	(* Internal method *)
	{attribute 'hide'}
	METHOD FB_init : BOOL
	VAR_INPUT
		(*  if TRUE, the retain variables are initialized (warm start / cold start) *)
		bInitRetains : BOOL;
		(*  if TRUE, the instance afterwards gets moved into the copy code (online change) *)
		bInCopyCode : BOOL;
	END_VAR
END_METHOD


	(* Internal method *)
	{attribute 'hide'}
	METHOD FB_exit : BOOL
	VAR_INPUT
		(*  if TRUE, the exit method is called for exiting an instance that is copied afterwards (online change). *)
		bInCopyCode : BOOL;
	END_VAR
END_METHOD


	(* Set the rotation angle in degrees [Â°]. *)
	METHOD SetAngle
	VAR_INPUT
		(* Rotation angle to set in degrees [Â°]. *)
		angle : LREAL;
	END_VAR
END_METHOD


	(* Set the components of this vector to '0.0'. *)
	METHOD SetZero
END_METHOD


	(* Set the components of this orientation. *)
	METHOD SetValues
	VAR_IN_OUT
		(* The position values to set. *)
 {attribute 'GUID' := 'ABCF5F54-5133-060C-4FEE-702387088411'}
				orientation2D : Orientation2D;
	END_VAR
END_METHOD


	(* Get the direction of the local x-axis. *)
	METHOD GetDirectionX
	VAR_IN_OUT
		(* The local x-direction of this orientation. *)
 {attribute 'GUID' := '619D5D7D-53EC-0B73-54D5-FB9C43AFDE82'}
				localX : TangentXY;
	END_VAR
END_METHOD


	(* Get the direction of the local y-axis. *)
	METHOD GetDirectionY
	VAR_IN_OUT
		(* The local y-direction of this orientation. *)
 {attribute 'GUID' := '619D5D7D-53EC-0B73-54D5-FB9C43AFDE82'}
				localY : TangentXY;
	END_VAR
END_METHOD


	(* Invert this position. *)
	METHOD Invert
END_METHOD


	(* Multiply an orientation to this orientation. *)
	METHOD ConcatenateWith
	VAR_IN_OUT
		(* Orientation to concatenate with. *)
 {attribute 'GUID' := 'ABCF5F54-5133-060C-4FEE-702387088411'}
				orientation2D : Orientation2D;
	END_VAR
END_METHOD


	(* Turn the orientation. *)
	METHOD TurnByC
	VAR_INPUT
		(* Rotation angle to turn by in degrees [Â°]. *)
		angle : LREAL;
	END_VAR
END_METHOD


	(* Rotate a PositionXY according to this orientation. *)
	METHOD Transform
	VAR_IN_OUT
		(* The orientation to multipy by. *)
 {attribute 'GUID' := 'D1D75488-37B1-0155-53AF-A9A9BDBB4FFD'}
				positionXY : PositionXY;
	END_VAR
END_METHOD


	PROPERTY angle : LREAL
GET
END_GET
SET
END_SET
END_PROPERTY

END_FUNCTION_BLOCK

// POUs/Spatial/Functions/ConcatenateABC

	{attribute 'TcIecLibraryType'}
	{attribute 'external_name' := 'ConcatenateABC_GUID_5F49A3AF_77BC_0B6E_5B9D_5571A51DBC7B'}
	(* Concatenate two instances of Orientation3D. *)
	FUNCTION ConcatenateABC : BOOL
	VAR_IN_OUT
		rotation0	:	Orientation3D;	(* 1st input orientation of the concatenation. *)
		rotation1	:	Orientation3D;	(* 2nd input orientation of the concatenation. *)
		concatenation	:	Orientation3D;	(* The concatenation of the two input instances. *)
	END_VAR

END_FUNCTION

// POUs/Spatial/Positions/Orientation3D

	{attribute 'c++_compatible'}
	{attribute 'external_name' := 'Orientation3D_GUID_CF039E61_7293_0F6E_5C80_E794F941E4DD'}
	{attribute 'TcIecLibraryType'}
	{attribute 'no_explicit_call' :='do not call this POU directly'}
	{attribute 'no_assign'}
	(* 3D orientation. All angles in degrees [Â°]. *)
	FUNCTION_BLOCK Orientation3D
	VAR
		(* Rotation around the 1st local axis in degrees [Â°]. *)
		p0 : LREAL;
		(* Rotation around 2nd local axis in degrees [Â°]. *)
		p1 : LREAL;
		(* Rotation around 3rd local axis in degrees [Â°]. *)
		p2 : LREAL;
		(* Defines the rotation order (rotate around local axes from left to right) *)
		 {attribute 'GUID' := 'BF8BCC1E-925E-4A57-801C-CC42AFDDA86D'}
		coordinates : E_RotationCoordinates := E_RotationCoordinates.CBA;
		 {attribute 'hide'}
		_reserved1 : ARRAY [1..84] OF USINT;
	END_VAR


	(* Internal method *)
	{attribute 'hide'}
	METHOD FB_init : BOOL
	VAR_INPUT
		(*  if TRUE, the retain variables are initialized (warm start / cold start) *)
		bInitRetains : BOOL;
		(*  if TRUE, the instance afterwards gets moved into the copy code (online change) *)
		bInCopyCode : BOOL;
	END_VAR
END_METHOD


	(* Internal method *)
	{attribute 'hide'}
	METHOD FB_exit : BOOL
	VAR_INPUT
		(*  if TRUE, the exit method is called for exiting an instance that is copied afterwards (online change). *)
		bInCopyCode : BOOL;
	END_VAR
END_METHOD


	(* Set the components of this vector to '0.0'. *)
	METHOD SetZero
END_METHOD


	(* Set the components of this position. *)
	METHOD SetValues
	VAR_IN_OUT
		(* The position values to set. *)
 {attribute 'GUID' := 'CF039E61-7293-0F6E-5C80-E794F941E4DD'}
				orientation3D : Orientation3D;
	END_VAR
END_METHOD


	(* Set the coordinates of the orientation. *)
	METHOD SetValuesABC
	VAR_INPUT
		(* 1st rotation angle in degrees [Â°]. *)
		phi0 : LREAL;
		(* 2nd rotation angle in degrees [Â°]. *)
		phi1 : LREAL;
		(* 3rd rotation angle in degrees [Â°]. *)
		phi2 : LREAL;
	END_VAR
END_METHOD


	(* Set the coordinates of the orientation. *)
	METHOD SetValuesACB
	VAR_INPUT
		(* 1st rotation angle in degrees [Â°]. *)
		phi0 : LREAL;
		(* 2nd rotation angle in degrees [Â°]. *)
		phi1 : LREAL;
		(* 3rd rotation angle in degrees [Â°]. *)
		phi2 : LREAL;
	END_VAR
END_METHOD


	(* Set the coordinates of the orientation. *)
	METHOD SetValuesBCA
	VAR_INPUT
		(* 1st rotation angle in degrees [Â°]. *)
		phi0 : LREAL;
		(* 2nd rotation angle in degrees [Â°]. *)
		phi1 : LREAL;
		(* 3rd rotation angle in degrees [Â°]. *)
		phi2 : LREAL;
	END_VAR
END_METHOD


	(* Set the coordinates of the orientation. *)
	METHOD SetValuesBAC
	VAR_INPUT
		(* 1st rotation angle in degrees [Â°]. *)
		phi0 : LREAL;
		(* 2nd rotation angle in degrees [Â°]. *)
		phi1 : LREAL;
		(* 3rd rotation angle in degrees [Â°]. *)
		phi2 : LREAL;
	END_VAR
END_METHOD


	(* Set the coordinates of the orientation. *)
	METHOD SetValuesCAB
	VAR_INPUT
		(* 1st rotation angle in degrees [Â°]. *)
		phi0 : LREAL;
		(* 2nd rotation angle in degrees [Â°]. *)
		phi1 : LREAL;
		(* 3rd rotation angle in degrees [Â°]. *)
		phi2 : LREAL;
	END_VAR
END_METHOD


	(* Set the coordinates of the orientation. *)
	METHOD SetValuesCBA
	VAR_INPUT
		(* 1st rotation angle in degrees [Â°]. *)
		phi0 : LREAL;
		(* 2nd rotation angle in degrees [Â°]. *)
		phi1 : LREAL;
		(* 3rd rotation angle in degrees [Â°]. *)
		phi2 : LREAL;
	END_VAR
END_METHOD


	(* Set the coordinates of the orientation. *)
	METHOD SetValuesABA
	VAR_INPUT
		(* 1st rotation angle in degrees [Â°]. *)
		phi0 : LREAL;
		(* 2nd rotation angle in degrees [Â°]. *)
		phi1 : LREAL;
		(* 3rd rotation angle in degrees [Â°]. *)
		phi2 : LREAL;
	END_VAR
END_METHOD


	(* Set the coordinates of the orientation. *)
	METHOD SetValuesACA
	VAR_INPUT
		(* 1st rotation angle in degrees [Â°]. *)
		phi0 : LREAL;
		(* 2nd rotation angle in degrees [Â°]. *)
		phi1 : LREAL;
		(* 3rd rotation angle in degrees [Â°]. *)
		phi2 : LREAL;
	END_VAR
END_METHOD


	(* Set the coordinates of the orientation. *)
	METHOD SetValuesBCB
	VAR_INPUT
		(* 1st rotation angle in degrees [Â°]. *)
		phi0 : LREAL;
		(* 2nd rotation angle in degrees [Â°]. *)
		phi1 : LREAL;
		(* 3rd rotation angle in degrees [Â°]. *)
		phi2 : LREAL;
	END_VAR
END_METHOD


	(* Set the coordinates of the orientation. *)
	METHOD SetValuesBAB
	VAR_INPUT
		(* 1st rotation angle in degrees [Â°]. *)
		phi0 : LREAL;
		(* 2nd rotation angle in degrees [Â°]. *)
		phi1 : LREAL;
		(* 3rd rotation angle in degrees [Â°]. *)
		phi2 : LREAL;
	END_VAR
END_METHOD


	(* Set the coordinates of the orientation. *)
	METHOD SetValuesCAC
	VAR_INPUT
		(* 1st rotation angle in degrees [Â°]. *)
		phi0 : LREAL;
		(* 2nd rotation angle in degrees [Â°]. *)
		phi1 : LREAL;
		(* 3rd rotation angle in degrees [Â°]. *)
		phi2 : LREAL;
	END_VAR
END_METHOD


	(* Set the coordinates of the orientation. *)
	METHOD SetValuesCBC
	VAR_INPUT
		(* 1st rotation angle in degrees [Â°]. *)
		phi0 : LREAL;
		(* 2nd rotation angle in degrees [Â°]. *)
		phi1 : LREAL;
		(* 3rd rotation angle in degrees [Â°]. *)
		phi2 : LREAL;
	END_VAR
END_METHOD


	(* Get the direction of the local x-axis. *)
	METHOD GetDirectionX
	VAR_IN_OUT
		(* The local x-direction of this orientation. *)
 {attribute 'GUID' := 'B2E383A0-A70D-05BB-6EF1-4EF1FE579E25'}
				localX : Tangent3D;
	END_VAR
END_METHOD


	(* Get the direction of the local y-axis. *)
	METHOD GetDirectionY
	VAR_IN_OUT
		(* The local y-direction of this orientation. *)
 {attribute 'GUID' := 'B2E383A0-A70D-05BB-6EF1-4EF1FE579E25'}
				localY : Tangent3D;
	END_VAR
END_METHOD


	(* Get the direction of the local z-axis. *)
	METHOD GetDirectionZ
	VAR_IN_OUT
		(* The local z-direction of this orientation. *)
 {attribute 'GUID' := 'B2E383A0-A70D-05BB-6EF1-4EF1FE579E25'}
				localZ : Tangent3D;
	END_VAR
END_METHOD


	(* Invert this position. *)
	METHOD Invert
END_METHOD


	(* Multiply an orientation to this orientation. *)
	METHOD ConcatenateWith
	VAR_IN_OUT
		(* Orientation to concatenate with. *)
 {attribute 'GUID' := 'CF039E61-7293-0F6E-5C80-E794F941E4DD'}
				orientation : Orientation3D;
	END_VAR
END_METHOD


	(* Rotate around an arbitrary local axis. The turn angle is given by the length of the axis. *)
	METHOD TurnBy
	VAR_IN_OUT
		(* The axis of rotation. Its length represents the angle of rotation in degrees [Â°]. *)
 {attribute 'GUID' := '40BB739E-8B51-070D-548D-A1BF22EE7364'}
				axis : TangentABC;
	END_VAR
END_METHOD


	(* Rotation around the local x-axis. *)
	METHOD TurnByA
	VAR_INPUT
		(* The angle to rotate by in degrees [Â°]. *)
		da : LREAL;
	END_VAR
END_METHOD


	(* Rotation around the local y-axis. *)
	METHOD TurnByB
	VAR_INPUT
		(* The angle to rotate by in degrees [Â°]. *)
		db : LREAL;
	END_VAR
END_METHOD


	(* Rotation around the local z-axis. *)
	METHOD TurnByC
	VAR_INPUT
		(* The angle to rotate by in degrees [Â°]. *)
		dc : LREAL;
	END_VAR
END_METHOD


	(* Rotate a Position3D according to this orientation. *)
	METHOD Transform
	VAR_IN_OUT
		(* Position to transform. *)
 {attribute 'GUID' := '6D9DE39A-582F-0FB5-796C-F5BBE97EF7B7'}
				position3D : Position3D;
	END_VAR
END_METHOD


	PROPERTY phi0 : LREAL
GET
END_GET
SET
END_SET
END_PROPERTY


	PROPERTY phi1 : LREAL
GET
END_GET
SET
END_SET
END_PROPERTY


	PROPERTY phi2 : LREAL
GET
END_GET
SET
END_SET
END_PROPERTY


	PROPERTY convention : E_RotationCoordinates
GET
END_GET
SET
END_SET
END_PROPERTY

END_FUNCTION_BLOCK

// POUs/Spatial/Functions/ConcatenateXYC

	{attribute 'TcIecLibraryType'}
	{attribute 'external_name' := 'ConcatenateXYC_GUID_78D6F5F6_2D9D_0BC8_5BA6_4CCA9448E29E'}
	(* Concatenate two instances of PositionXYC. *)
	FUNCTION ConcatenateXYC : BOOL
	VAR_IN_OUT
		position0	:	PositionXYC;	(* 1st input position of the concatenation. *)
		position1	:	PositionXYC;	(* 2nd input position of the concatenation. *)
		concatenation	:	PositionXYC;	(* The concatenation of the two input instances. *)
	END_VAR

END_FUNCTION

// POUs/Spatial/Functions/Concatenate6D

	{attribute 'TcIecLibraryType'}
	{attribute 'external_name' := 'Concatenate6D_GUID_8EBEEF7C_23E7_0FBE_6933_AD0676D13CAF'}
	(* Concatenate two instances of PositionSE3. *)
	FUNCTION Concatenate6D : BOOL
	VAR_IN_OUT
		position0	:	PositionSE3;	(* 1st input position of the concatenation. *)
		position1	:	PositionSE3;	(* 2nd input position of the concatenation. *)
		concatenation	:	PositionXYC;	(* The concatenation of the two input instances. *)
	END_VAR

END_FUNCTION

// POUs/Spatial/Functions/AddXY

	{attribute 'TcIecLibraryType'}
	{attribute 'external_name' := 'AddXY_GUID_DDD35889_D84D_05EB_6F65_1B96CF5EB621'}
	(* Add two instances of TangentXY. *)
	FUNCTION AddXY : BOOL
	VAR_IN_OUT
		tangent0	:	TangentXY;	(* 1st input tangent vector. *)
		tangent1	:	TangentXY;	(* 2nd input tangent vector. *)
		sumTangent	:	TangentXY;	(* Sum of the two tangent vectors. *)
	END_VAR

END_FUNCTION

// POUs/Spatial/Functions/SubtractXY

	{attribute 'TcIecLibraryType'}
	{attribute 'external_name' := 'SubtractXY_GUID_0C6F5B78_D359_0731_5E59_E056E947D4D6'}
	(* Subtract two instances of TangentXY. *)
	FUNCTION SubtractXY : BOOL
	VAR_IN_OUT
		tangent0	:	TangentXY;	(* 1st input tangent vector. *)
		tangent1	:	TangentXY;	(* 2nd input tangent vector. *)
		difference	:	TangentXY;	(* Difference of the two tangent vectors. *)
	END_VAR

END_FUNCTION

// POUs/Spatial/Functions/MultiplyXY

	{attribute 'TcIecLibraryType'}
	{attribute 'external_name' := 'MultiplyXY_GUID_C2C4AD6C_C4AC_0794_59D0_610FF6034C86'}
	(* Multiply a TangentXY by a scalar and return the result. *)
	FUNCTION MultiplyXY : BOOL
	VAR_IN_OUT
		tangent	:	TangentXY;	(* Tangent vector to multiply. *)
	END_VAR
	VAR_INPUT
		scalar	:	LREAL;	(* Scalar value to multiply with. *)
	END_VAR
	VAR_IN_OUT
		scaled	:	TangentXY;	(* Scaled input tangent vector. *)
	END_VAR

END_FUNCTION

// POUs/Spatial/Functions/ScalarXY

	{attribute 'TcIecLibraryType'}
	{attribute 'external_name' := 'ScalarXY_GUID_D4D96D10_2A9C_014D_517A_5634DCDE2F41'}
	(* Compute the scalar product of two instance of TangentXY. *)
	FUNCTION ScalarXY : LREAL
	VAR_IN_OUT
		tangent0	:	TangentXY;	(* 1st input tangent vector. *)
		tangent1	:	TangentXY;	(* 2nd input tangent vector. *)
	END_VAR

END_FUNCTION

// POUs/Spatial/Functions/Add3D

	{attribute 'TcIecLibraryType'}
	{attribute 'external_name' := 'Add3D_GUID_1E13EC6A_6354_0916_764A_72852C2363FA'}
	(* Add two instances of Tangent3D. *)
	FUNCTION Add3D : BOOL
	VAR_IN_OUT
		tangent0	:	Tangent3D;	(* 1st input tangent vector. *)
		tangent1	:	Tangent3D;	(* 2nd input tangent vector. *)
		sumTangent	:	Tangent3D;	(* Sum of the two tangent vectors. *)
	END_VAR

END_FUNCTION

// POUs/Spatial/Functions/Subtract3D

	{attribute 'TcIecLibraryType'}
	{attribute 'external_name' := 'Subtract3D_GUID_03B5443E_D84E_0CB8_5880_268654118928'}
	(* Subtract two instances of Tangent3D. *)
	FUNCTION Subtract3D : BOOL
	VAR_IN_OUT
		tangent0	:	Tangent3D;	(* 1st input tangent vector. *)
		tangent1	:	Tangent3D;	(* 2nd input tangent vector. *)
		difference	:	Tangent3D;	(* Difference of the two tangent vectors. *)
	END_VAR

END_FUNCTION

// POUs/Spatial/Functions/Multiply3D

	{attribute 'TcIecLibraryType'}
	{attribute 'external_name' := 'Multiply3D_GUID_7F10E0AD_D224_08E4_56FE_84A3CADD7D2A'}
	(* Multiply a Tangent3D by a scalar. *)
	FUNCTION Multiply3D : BOOL
	VAR_IN_OUT
		tangent	:	Tangent3D;	(* Tangent vector to multiply. *)
	END_VAR
	VAR_INPUT
		scalar	:	LREAL;	(* Scalar value to multiply with. *)
	END_VAR
	VAR_IN_OUT
		scaled	:	Tangent3D;	(* Scaled input tangent vector. *)
	END_VAR

END_FUNCTION

// POUs/Spatial/Functions/Scalar3D

	{attribute 'TcIecLibraryType'}
	{attribute 'external_name' := 'Scalar3D_GUID_8AF04058_8F46_0BFD_4BB7_03B3239446C2'}
	(* Compute the scalar product of two instances of Tangent3D. *)
	FUNCTION Scalar3D : LREAL
	VAR_IN_OUT
		tangent0	:	Tangent3D;	(* 1st input tangent vector. *)
		tangent1	:	Tangent3D;	(* 2nd input tangent vector. *)
	END_VAR

END_FUNCTION

// POUs/Spatial/Functions/Cross3D

	{attribute 'TcIecLibraryType'}
	{attribute 'external_name' := 'Cross3D_GUID_5FD8B2DF_C59D_0830_7394_4BAB2DFF32FF'}
	(* Compute the cross product of two instances of Tangent3D. *)
	FUNCTION Cross3D : BOOL
	VAR_IN_OUT
		tangent0	:	Tangent3D;	(* 1st input tangent vector. *)
		tangent1	:	Tangent3D;	(* 2nd input tangent vector. *)
		crossProduct	:	Tangent3D;	(* The resulting cross product. *)
	END_VAR

END_FUNCTION

// POUs/Spatial/Functions/AddABC

	{attribute 'TcIecLibraryType'}
	{attribute 'external_name' := 'AddABC_GUID_8FDE7604_65CA_062E_690C_F9BF9E165754'}
	(* Add two instances of TangentABC. *)
	FUNCTION AddABC : BOOL
	VAR_IN_OUT
		tangent0	:	TangentABC;	(* 1st input tangent vector. *)
		tangent1	:	TangentABC;	(* 2nd input tangent vector. *)
		sumTangent	:	TangentABC;	(* Sum of the two tangent vectors. *)
	END_VAR

END_FUNCTION

// POUs/Spatial/Functions/SubtractABC

	{attribute 'TcIecLibraryType'}
	{attribute 'external_name' := 'SubtractABC_GUID_3261EE05_4E2C_04FD_5CF9_C86591DE64D1'}
	(* Subtract two instances of TangentABC. *)
	FUNCTION SubtractABC : BOOL
	VAR_IN_OUT
		tangent0	:	TangentABC;	(* 1st input tangent vector. *)
		tangent1	:	TangentABC;	(* 2nd input tangent vector. *)
		difference	:	TangentABC;	(* Difference of the two tangent vectors. *)
	END_VAR

END_FUNCTION

// POUs/Spatial/Functions/MultiplyABC

	{attribute 'TcIecLibraryType'}
	{attribute 'external_name' := 'MultiplyABC_GUID_F273EF0A_B0F2_0BB8_4B63_CA32C22A9DFF'}
	(* Multiply a TangentABC by a scalar. *)
	FUNCTION MultiplyABC : BOOL
	VAR_IN_OUT
		tangent	:	TangentABC;	(* Tangent vector to multiply. *)
	END_VAR
	VAR_INPUT
		scalar	:	LREAL;	(* Scalar value to multiply with. *)
	END_VAR
	VAR_IN_OUT
		scaled	:	TangentABC;	(* Scaled input tangent vector. *)
	END_VAR

END_FUNCTION

// POUs/Spatial/Functions/AddXYC

	{attribute 'TcIecLibraryType'}
	{attribute 'external_name' := 'AddXYC_GUID_22B2DB7F_2171_0022_56E0_856985EACA76'}
	(* Add two instances of TangentXYC. *)
	FUNCTION AddXYC : BOOL
	VAR_IN_OUT
		tangent0	:	TangentXYC;	(* 1st input tangent vector. *)
		tangent1	:	TangentXYC;	(* 2nd input tangent vector. *)
		sumTangent	:	TangentXYC;	(* Sum of the two tangent vectors. *)
	END_VAR

END_FUNCTION

// POUs/Spatial/Functions/SubtractXYC

	{attribute 'TcIecLibraryType'}
	{attribute 'external_name' := 'SubtractXYC_GUID_E14F8DE0_72BF_0E78_69F5_065A37DBA031'}
	(* Subtract two instances of TangentXYC. *)
	FUNCTION SubtractXYC : BOOL
	VAR_IN_OUT
		tangent0	:	TangentXYC;	(* 1st input tangent vector. *)
		tangent1	:	TangentXYC;	(* 2nd input tangent vector. *)
		difference	:	TangentXYC;	(* Difference of the two tangent vectors. *)
	END_VAR

END_FUNCTION

// POUs/Spatial/Functions/MultiplyXYC

	{attribute 'TcIecLibraryType'}
	{attribute 'external_name' := 'MultiplyXYC_GUID_579519F2_727C_050B_6CC1_FDCF5EF7A66B'}
	(* Multiply a TangentXYC by a scalar. *)
	FUNCTION MultiplyXYC : BOOL
	VAR_IN_OUT
		tangent	:	TangentXYC;	(* Tangent vector to multiply. *)
	END_VAR
	VAR_INPUT
		scalar	:	LREAL;	(* Scalar value to multiply with. *)
	END_VAR
	VAR_IN_OUT
		scaled	:	TangentXYC;	(* Scaled input tangent vector. *)
	END_VAR

END_FUNCTION

// POUs/Spatial/Functions/Add6D

	{attribute 'TcIecLibraryType'}
	{attribute 'external_name' := 'Add6D_GUID_37B28D4C_24D7_0C0E_5B06_85D7BA99C789'}
	(* Add two instances of Tangent6D. *)
	FUNCTION Add6D : BOOL
	VAR_IN_OUT
		tangent0	:	Tangent6D;	(* 1st input tangent vector. *)
		tangent1	:	Tangent6D;	(* 2nd input tangent vector. *)
		sumTangent	:	Tangent6D;	(* Sum of the two tangent vectors. *)
	END_VAR

END_FUNCTION

// POUs/Spatial/Functions/Subtract6D

	{attribute 'TcIecLibraryType'}
	{attribute 'external_name' := 'Subtract6D_GUID_C221F786_39D2_03E1_7E75_787679E49BC2'}
	(* Subtract two instances of Tangent6D. *)
	FUNCTION Subtract6D : BOOL
	VAR_IN_OUT
		tangent0	:	Tangent6D;	(* 1st input tangent vector. *)
		tangent1	:	Tangent6D;	(* 2nd input tangent vector. *)
		difference	:	Tangent6D;	(* Difference of the two tangent vectors. *)
	END_VAR

END_FUNCTION

// POUs/Spatial/Functions/Multiply6D

	{attribute 'TcIecLibraryType'}
	{attribute 'external_name' := 'Multiply6D_GUID_D67C9F17_5B6C_000C_64F8_8CE8AE9429C6'}
	(* Multiply a Tangent6D by a scalar. *)
	FUNCTION Multiply6D : BOOL
	VAR_IN_OUT
		tangent	:	Tangent6D;	(* Tangent vector to multiply. *)
	END_VAR
	VAR_INPUT
		scalar	:	LREAL;	(* Scalar value to multiply with. *)
	END_VAR
	VAR_IN_OUT
		scaled	:	Tangent6D;	(* Scaled input tangent vector. *)
	END_VAR

END_FUNCTION

// POUs/Spatial/Functions/ConvertToCartesian2D

	{attribute 'TcIecLibraryType'}
	{attribute 'external_name' := 'ConvertToCartesian2D_GUID_5AC5CB59_5367_097E_5B20_94D940232A25'}
	(* Convert local XYC-dynamic properties to global XY ones. *)
	FUNCTION ConvertToCartesian2D : BOOL
	VAR_IN_OUT
		position	:	PositionXYC;	(* The position hosting the local dynamic state. *)
		velocity	:	TangentXYC;	(* The local velocity vector. *)
		acceleration	:	TangentXYC;	(* The local acceleration vector. *)
		velocity_XY	:	TangentXY;	(* The resulting global Cartesian velocity. *)
		acceleration_XY	:	TangentXY;	(* The resulting global Cartesian acceleration. *)
	END_VAR

END_FUNCTION

// POUs/Spatial/Setpoints/SetpointR1

	{attribute 'c++_compatible'}
	{attribute 'external_name' := 'SetpointR1_GUID_0BDDEBC9_5233_0AE3_6BFE_B96BF70FB5CC'}
	{attribute 'TcIecLibraryType'}
	{attribute 'no_explicit_call' :='do not call this POU directly'}
	{attribute 'no_assign_warning'}
	(* 1D setpoint. *)
	FUNCTION_BLOCK SetpointR1
	VAR
		(* Position component of the setpoint. *)
		ds : LREAL;
		(* Velocity component of the setpoint. *)
		dv : LREAL;
		(* Acceleration component of the setpoint. *)
		da : LREAL;
		(* Jerk component of the setpoint. *)
		dj : LREAL;
	END_VAR


	(* Internal method *)
	{attribute 'hide'}
	METHOD FB_init : BOOL
	VAR_INPUT
		(*  if TRUE, the retain variables are initialized (warm start / cold start) *)
		bInitRetains : BOOL;
		(*  if TRUE, the instance afterwards gets moved into the copy code (online change) *)
		bInCopyCode : BOOL;
	END_VAR
END_METHOD


	(* Internal method *)
	{attribute 'hide'}
	METHOD FB_reinit : BOOL
END_METHOD


	(* Internal method *)
	{attribute 'hide'}
	METHOD FB_exit : BOOL
	VAR_INPUT
		(*  if TRUE, the exit method is called for exiting an instance that is copied afterwards (online change). *)
		bInCopyCode : BOOL;
	END_VAR
END_METHOD


	(* Set this setpoint to zero. *)
	METHOD SetZero
END_METHOD


	(* Set the values of this coordinate. *)
	METHOD SetValuesSVAJ
	VAR_INPUT
		(* the position value to set. *)
		_s : LREAL;
		(* the velocity value to set. *)
		v : LREAL;
		(* the acceleration value to set. *)
		a : LREAL;
		(* the jerk value to set. *)
		j : LREAL;
	END_VAR
END_METHOD


	PROPERTY _s : LREAL
GET
END_GET
SET
END_SET
END_PROPERTY


	PROPERTY v : LREAL
GET
END_GET
SET
END_SET
END_PROPERTY


	PROPERTY a : LREAL
GET
END_GET
SET
END_SET
END_PROPERTY


	PROPERTY j : LREAL
GET
END_GET
SET
END_SET
END_PROPERTY

END_FUNCTION_BLOCK

// POUs/Spatial/Setpoints/SetpointSE3

	{attribute 'c++_compatible'}
	{attribute 'external_name' := 'SetpointSE3_GUID_9F524B81_AD7E_028A_4B16_31B8A72EF3B3'}
	{attribute 'TcIecLibraryType'}
	{attribute 'no_explicit_call' :='do not call this POU directly'}
	{attribute 'no_assign_warning'}
	(* SE3 setpoint. *)
	FUNCTION_BLOCK SetpointSE3 EXTENDS IPlcGeometry3D


	(* Internal method *)
	{attribute 'hide'}
	METHOD FB_init : BOOL
	VAR_INPUT
		(*  if TRUE, the retain variables are initialized (warm start / cold start) *)
		bInitRetains : BOOL;
		(*  if TRUE, the instance afterwards gets moved into the copy code (online change) *)
		bInCopyCode : BOOL;
	END_VAR
END_METHOD


	(* Internal method *)
	{attribute 'hide'}
	METHOD FB_exit : BOOL
	VAR_INPUT
		(*  if TRUE, the exit method is called for exiting an instance that is copied afterwards (online change). *)
		bInCopyCode : BOOL;
	END_VAR
END_METHOD


	(* Set this setpoint to be the identity. *)
	METHOD SetIdentity
END_METHOD


	(* Set the values of this setpoint. *)
	METHOD SetValues
	VAR_IN_OUT
		(* The setpoint to copy. *)
 {attribute 'GUID' := '9F524B81-AD7E-028A-4B16-31B8A72EF3B3'}
				setpoint : SetpointSE3;
	END_VAR
END_METHOD


	(* Set the cartesian values of this setpoint. *)
	METHOD SetValuesXYZ
	VAR_IN_OUT
		(* The x-setpoint to set. *)
 {attribute 'GUID' := '0BDDEBC9-5233-0AE3-6BFE-B96BF70FB5CC'}
				setpointX : SetpointR1;
		(* The y-setpoint to set. *)
 {attribute 'GUID' := '0BDDEBC9-5233-0AE3-6BFE-B96BF70FB5CC'}
				setpointY : SetpointR1;
		(* The z-setpoint to set. *)
 {attribute 'GUID' := '0BDDEBC9-5233-0AE3-6BFE-B96BF70FB5CC'}
				setpointZ : SetpointR1;
	END_VAR
END_METHOD


	(* Set the angular values of this setpoint. *)
	METHOD SetValuesCBA
	VAR_IN_OUT
		(* The c-setpoint to set. *)
 {attribute 'GUID' := '0BDDEBC9-5233-0AE3-6BFE-B96BF70FB5CC'}
				setpointC : SetpointR1;
		(* The b-setpoint to set. *)
 {attribute 'GUID' := '0BDDEBC9-5233-0AE3-6BFE-B96BF70FB5CC'}
				setpointB : SetpointR1;
		(* The a-setpoint to set. *)
 {attribute 'GUID' := '0BDDEBC9-5233-0AE3-6BFE-B96BF70FB5CC'}
				setpointA : SetpointR1;
	END_VAR
END_METHOD


	(* Get the direction of the local x-axis. *)
	METHOD GetDirectionX
	VAR_IN_OUT
		(* The local x-direction of this orientation. *)
 {attribute 'GUID' := 'B2E383A0-A70D-05BB-6EF1-4EF1FE579E25'}
				localX : Tangent3D;
	END_VAR
END_METHOD


	(* Get the direction of the local y-axis. *)
	METHOD GetDirectionY
	VAR_IN_OUT
		(* The local y-direction of this orientation. *)
 {attribute 'GUID' := 'B2E383A0-A70D-05BB-6EF1-4EF1FE579E25'}
				localY : Tangent3D;
	END_VAR
END_METHOD


	(* Get the direction of the local z-axis. *)
	METHOD GetDirectionZ
	VAR_IN_OUT
		(* The local z-direction of this orientation. *)
 {attribute 'GUID' := 'B2E383A0-A70D-05BB-6EF1-4EF1FE579E25'}
				localZ : Tangent3D;
	END_VAR
END_METHOD


	(* Get the linear Cartesian position components. *)
	METHOD GetPosition_Cartesian
	VAR_IN_OUT
		(* The output position. *)
 {attribute 'GUID' := '6D9DE39A-582F-0FB5-796C-F5BBE97EF7B7'}
				position : Position3D;
	END_VAR
END_METHOD


	(* Get the linear Cartesian velocity components. *)
	METHOD GetVelocity_Cartesian
	VAR_IN_OUT
		(* The output tangent. *)
 {attribute 'GUID' := 'B2E383A0-A70D-05BB-6EF1-4EF1FE579E25'}
				tangent : Tangent3D;
	END_VAR
END_METHOD


	(* Get the linear Cartesian acceleration components. *)
	METHOD GetAcceleration_Cartesian
	VAR_IN_OUT
		(* The output tangent. *)
 {attribute 'GUID' := 'B2E383A0-A70D-05BB-6EF1-4EF1FE579E25'}
				tangent : Tangent3D;
	END_VAR
END_METHOD


	(* Get the linear Cartesian jerk components. *)
	METHOD GetJerk_Cartesian
	VAR_IN_OUT
		(* The output tangent. *)
 {attribute 'GUID' := 'B2E383A0-A70D-05BB-6EF1-4EF1FE579E25'}
				tangent : Tangent3D;
	END_VAR
END_METHOD


	(* Concatenate this setpoint with a second one up to a specific order. *)
	METHOD ConcatenateWith
	VAR_IN_OUT
		(* The setpoint to concatenate. *)
 {attribute 'GUID' := '9F524B81-AD7E-028A-4B16-31B8A72EF3B3'}
				setpoint : SetpointSE3;
	END_VAR
	VAR_INPUT
		(*  The order up to which to compute. *)
		order : UDINT;
	END_VAR
END_METHOD


	PROPERTY x : LREAL
GET
END_GET
SET
END_SET
END_PROPERTY


	PROPERTY y : LREAL
GET
END_GET
SET
END_SET
END_PROPERTY


	PROPERTY z : LREAL
GET
END_GET
SET
END_SET
END_PROPERTY


	PROPERTY phi0 : LREAL
GET
END_GET
SET
END_SET
END_PROPERTY


	PROPERTY phi1 : LREAL
GET
END_GET
SET
END_SET
END_PROPERTY


	PROPERTY phi2 : LREAL
GET
END_GET
SET
END_SET
END_PROPERTY


	PROPERTY Convention : E_RotationCoordinates
GET
END_GET
SET
END_SET
END_PROPERTY

END_FUNCTION_BLOCK

// POUs/Spatial/Inertias/InertiaSE3

	{attribute 'c++_compatible'}
	{attribute 'external_name' := 'InertiaSE3_GUID_070343EC_747B_0B38_64A8_5FFF96978D36'}
	{attribute 'TcIecLibraryType'}
	{attribute 'no_explicit_call' :='do not call this POU directly'}
	{attribute 'no_assign'}
	(* Inertia tensor containing angular and linear inertia. *)
	FUNCTION_BLOCK InertiaSE3
	VAR
		(* Mass of the inertia. *)
		m : LREAL;
		(* x-component of the center of mass. *)
		CenterX : LREAL;
		(* y-component of the center of mass. *)
		CenterY : LREAL;
		(* z-component of the center of mass. *)
		CenterZ : LREAL;
		 {attribute 'hide'}
		_reserved1 : ARRAY [1..80] OF USINT;
	END_VAR


	(* Internal method *)
	{attribute 'hide'}
	METHOD FB_init : BOOL
	VAR_INPUT
		(*  if TRUE, the retain variables are initialized (warm start / cold start) *)
		bInitRetains : BOOL;
		(*  if TRUE, the instance afterwards gets moved into the copy code (online change) *)
		bInCopyCode : BOOL;
	END_VAR
END_METHOD


	(* Internal method *)
	{attribute 'hide'}
	METHOD FB_exit : BOOL
	VAR_INPUT
		(*  if TRUE, the exit method is called for exiting an instance that is copied afterwards (online change). *)
		bInCopyCode : BOOL;
	END_VAR
END_METHOD


	(* Add a 2nd inertia tensor to this one. *)
	METHOD AddBy
	VAR_IN_OUT
		(* The inertia tensor to add. *)
 {attribute 'GUID' := '070343EC-747B-0B38-64A8-5FFF96978D36'}
				shift : InertiaSE3;
	END_VAR
END_METHOD


	(* Set the values to that of a point. *)
	METHOD SetValues_Point
	VAR_INPUT
		(* The mass of the point. *)
		mass : LREAL;
		(* The x-position of the point. *)
		x : LREAL;
		(* The y-position of the point. *)
		y : LREAL;
		(* The z-position of the point. *)
		z : LREAL;
	END_VAR
END_METHOD


	(* Set the values to that of a sphere. *)
	METHOD SetValues_Sphere
	VAR_INPUT
		(* The mass of the sphere. *)
		mass : LREAL;
		(* The radius of the sphere. *)
		radius : LREAL;
	END_VAR
END_METHOD


	(* Set the values to that of a cylinder. *)
	METHOD SetValues_Cylinder
	VAR_INPUT
		(* The mass of the cylinder. *)
		mass : LREAL;
		(* The radius of the cylinder. *)
		radius : LREAL;
		(* The height of the cylinder. *)
		height : LREAL;
	END_VAR
END_METHOD


	(* Set the values to that of a cuboid. *)
	METHOD SetValues_Cuboid
	VAR_INPUT
		(* The mass of the cuboid. *)
		mass : LREAL;
		(* The x-length of the cuboid. *)
		dx : LREAL;
		(* The y-length of the cuboid. *)
		dy : LREAL;
		(* The z-length of the cuboid. *)
		dz : LREAL;
	END_VAR
END_METHOD


	(* Transform this inertia by a displacement. *)
	METHOD Transform
	VAR_IN_OUT
		(* The displacement to apply. *)
 {attribute 'GUID' := '4DF191CB-C971-05F9-659B-EBBADE382F22'}
				displacement : PositionSE3;
	END_VAR
END_METHOD


	(* Translate this inertia by a translation. *)
	METHOD Translate
	VAR_IN_OUT
		(* The translation to apply. *)
 {attribute 'GUID' := 'B2E383A0-A70D-05BB-6EF1-4EF1FE579E25'}
				displacement : Tangent3D;
	END_VAR
END_METHOD


	PROPERTY mass : LREAL
GET
END_GET
SET
END_SET
END_PROPERTY


	PROPERTY x : LREAL
GET
END_GET
SET
END_SET
END_PROPERTY


	PROPERTY y : LREAL
GET
END_GET
SET
END_SET
END_PROPERTY


	PROPERTY z : LREAL
GET
END_GET
SET
END_SET
END_PROPERTY


	PROPERTY xx : LREAL
GET
END_GET
SET
END_SET
END_PROPERTY


	PROPERTY yy : LREAL
GET
END_GET
SET
END_SET
END_PROPERTY


	PROPERTY zz : LREAL
GET
END_GET
SET
END_SET
END_PROPERTY


	PROPERTY xy : LREAL
GET
END_GET
SET
END_SET
END_PROPERTY


	PROPERTY yz : LREAL
GET
END_GET
SET
END_SET
END_PROPERTY


	PROPERTY zx : LREAL
GET
END_GET
SET
END_SET
END_PROPERTY

END_FUNCTION_BLOCK

// POUs/Shapes/Geometry2D/Container2D

	{attribute 'c++_compatible'}
	{attribute 'external_name' := 'Container2D_GUID_767E92D3_F6C2_0661_63DA_E22E4121F453'}
	{attribute 'TcIecLibraryType'}
	{attribute 'no_explicit_call' :='do not call this POU directly'}
	{attribute 'no_assign'}
	FUNCTION_BLOCK Container2D EXTENDS Geometry2D


	(* Internal method *)
	METHOD FB_init : BOOL
	VAR_INPUT
		(*  if TRUE, the retain variables are initialized (warm start / cold start) *)
		bInitRetains : BOOL;
		(*  if TRUE, the instance afterwards gets moved into the copy code (online change) *)
		bInCopyCode : BOOL;
	END_VAR
END_METHOD


	(* Internal method *)
	{attribute 'hide'}
	METHOD FB_exit : BOOL
	VAR_INPUT
		(*  if TRUE, the exit method is called for exiting an instance that is copied afterwards (online change). *)
		bInCopyCode : BOOL;
	END_VAR
END_METHOD


	(* Add a geometry to the container. *)
	METHOD AddElement : UDINT
	VAR_IN_OUT
		(* The geometry to add. *)
 {attribute 'GUID' := 'EA1925AE-2507-0F27-40AC-5A565B8F6BBE'}
				inputObject : Geometry2D;
	END_VAR
END_METHOD


	(* Remove a specified geometry from the container. *)
	METHOD RemoveElement
	VAR_INPUT
		(* ID of the geometry to remove. *)
		id : UDINT;
	END_VAR
END_METHOD


	(* Remove all geometries from the container. *)
	METHOD Clear
END_METHOD


	(* Get the number of geometry elements in container. *)
	METHOD GetCount : UDINT
END_METHOD


	(* Get the combined boundary of all hosted 2D-geometries. *)
	METHOD GetBoundary
	VAR_IN_OUT
		(* The combined boundary.. *)
 {attribute 'GUID' := '767E92D3-F6C2-0661-63DA-E22E4121F453'}
				boundary : Container2D;
	END_VAR
END_METHOD

END_FUNCTION_BLOCK

// POUs/Shapes/Geometry2D/Extrude2D

	{attribute 'c++_compatible'}
	{attribute 'external_name' := 'Extrude2D_GUID_E01C1478_0DB7_05D8_6DD0_7ED3D5C1A09A'}
	{attribute 'TcIecLibraryType'}
	{attribute 'no_explicit_call' :='do not call this POU directly'}
	{attribute 'no_assign'}
	FUNCTION_BLOCK Extrude2D EXTENDS Geometry2D


	(* Internal method *)
	METHOD FB_init : BOOL
	VAR_INPUT
		(*  if TRUE, the retain variables are initialized (warm start / cold start) *)
		bInitRetains : BOOL;
		(*  if TRUE, the instance afterwards gets moved into the copy code (online change) *)
		bInCopyCode : BOOL;
	END_VAR
END_METHOD


	(* Internal method *)
	{attribute 'hide'}
	METHOD FB_exit : BOOL
	VAR_INPUT
		(*  if TRUE, the exit method is called for exiting an instance that is copied afterwards (online change). *)
		bInCopyCode : BOOL;
	END_VAR
END_METHOD


	(* Define the extrusion geometry by a path and the corners to extrude. *)
	METHOD ExtrudeAlong
	VAR_IN_OUT
		(* The path to extrude along. *)
 {attribute 'GUID' := '43690AE8-9937-053A-4530-699ADF0ABACD'}
				path : PathXYC;
	END_VAR
	VAR_INPUT
		(* 1st distance from the path to extrude. *)
		dy0 : LREAL;
		(* 2nd distance from the path to extrude. *)
		dy1 : LREAL;
		(* Number of steps to employ along the path. *)
		extrusionSteps : UDINT;
	END_VAR
END_METHOD


	(* Check whether this extrusion geometry is valid. *)
	METHOD IsValid : BOOL
END_METHOD

END_FUNCTION_BLOCK

// POUs/Paths/Components/PathXYC

	{attribute 'c++_compatible'}
	{attribute 'external_name' := 'PathXYC_GUID_43690AE8_9937_053A_4530_699ADF0ABACD'}
	{attribute 'TcIecLibraryType'}
	{attribute 'no_explicit_call' :='do not call this POU directly'}
	{attribute 'no_assign'}
	(* A path in the xy-plane with an additional orientation at every path position. *)
	FUNCTION_BLOCK PathXYC EXTENDS IPlcPath2D


	(* Internal method *)
	{attribute 'hide'}
	METHOD FB_init : BOOL
	VAR_INPUT
		(*  if TRUE, the retain variables are initialized (warm start / cold start) *)
		bInitRetains : BOOL;
		(*  if TRUE, the instance afterwards gets moved into the copy code (online change) *)
		bInCopyCode : BOOL;
	END_VAR
END_METHOD


	(* Internal method *)
	{attribute 'hide'}
	METHOD FB_exit : BOOL
	VAR_INPUT
		(*  if TRUE, the exit method is called for exiting an instance that is copied afterwards (online change). *)
		bInCopyCode : BOOL;
	END_VAR
END_METHOD


	(* Append a smooth transition from the current end of the path
				    to the specified position. *)
	METHOD AppendPosition
	VAR_IN_OUT
		(* The position to append. *)
 {attribute 'GUID' := '54EDED35-5A53-0913-4680-EA5D332AAA4F'}
				position : PositionXYC;
	END_VAR
END_METHOD


	(* Append a smooth transition from the current end of the path
				    to the specified position. *)
	METHOD AppendPositionXYC
	VAR_INPUT
		(* x-component of the position to append. *)
		x : LREAL;
		(* y-component of the position to append. *)
		y : LREAL;
		(* c-component of the position to append in degrees [Â°]. *)
		c : LREAL;
	END_VAR
END_METHOD


	(* Append a line to this path. *)
	METHOD AppendLine
	VAR_IN_OUT
		(* Start position of the line. *)
 {attribute 'GUID' := '54EDED35-5A53-0913-4680-EA5D332AAA4F'}
				startPos : PositionXYC;
		(* End position of the line. *)
 {attribute 'GUID' := '54EDED35-5A53-0913-4680-EA5D332AAA4F'}
				endPos : PositionXYC;
	END_VAR
END_METHOD


	(* Append a circle to this path. *)
	METHOD AppendCircle
	VAR_IN_OUT
		(* Start position of the circle. *)
 {attribute 'GUID' := '54EDED35-5A53-0913-4680-EA5D332AAA4F'}
				startPos : PositionXYC;
		(* End position of the circle. *)
 {attribute 'GUID' := '54EDED35-5A53-0913-4680-EA5D332AAA4F'}
				endPos : PositionXYC;
		(* Center of the circle. *)
 {attribute 'GUID' := 'D1D75488-37B1-0155-53AF-A9A9BDBB4FFD'}
				center : PositionXY;
	END_VAR
	VAR_INPUT
		(* Set whether the circle runs clockwise or counter-clockwise. *)
		clockwise : BOOL;
	END_VAR
END_METHOD


	(* Appends a smooth transition from the end of this path
				      to the start of the other path, locking further changes of this path. *)
	METHOD EndAtPath
	VAR_IN_OUT
		(* The other path. *)
 {attribute 'GUID' := '43690AE8-9937-053A-4530-699ADF0ABACD'}
				path : PathXYC;
	END_VAR
END_METHOD


	(* Appends a smooth transition from the start of this path
				      to the end of the other path, locking further changes of the other path. *)
	METHOD StartFromPath
	VAR_IN_OUT
		(* The other path. *)
 {attribute 'GUID' := '43690AE8-9937-053A-4530-699ADF0ABACD'}
				path : PathXYC;
	END_VAR
END_METHOD


	(* Connect start and end position.
				      A smooth transition is added as long as start and end positin are not identical.
				      This operation finalizes this path definition and locks it against further modifications. *)
	METHOD CloseLoop
END_METHOD


	(* Empty all current path definitions and reset the path back to an empty state. *)
	METHOD Clear
END_METHOD


	(* Get the start position of the path. *)
	METHOD GetStartPosition
	VAR_IN_OUT
		(* The current start position of the path. *)
 {attribute 'GUID' := '54EDED35-5A53-0913-4680-EA5D332AAA4F'}
				startPosition : PositionXYC;
	END_VAR
END_METHOD


	(* Get the end position of the segment. *)
	METHOD GetEndPosition
	VAR_IN_OUT
		(* The current end position of the segment. *)
 {attribute 'GUID' := '54EDED35-5A53-0913-4680-EA5D332AAA4F'}
				endPosition : PositionXYC;
	END_VAR
END_METHOD


	(* Get a position on the path at a specific arclength value. *)
	METHOD GetPositionAt
	VAR_INPUT
		(* Arc length value where the position is evaluated. *)
		arcLength : LREAL;
	END_VAR
	VAR_IN_OUT
		(* The position at the specified arc parameter. *)
 {attribute 'GUID' := '54EDED35-5A53-0913-4680-EA5D332AAA4F'}
				position : PositionXYC;
	END_VAR
END_METHOD


	(* Get the dynamic information when moving along a path
				    with specific arclength value and dynamic changes. *)
	METHOD GetStateAt
	VAR_INPUT
		(* Arc length value where the position is evaluated. *)
		arcLength : LREAL;
		(* Velocity of the arc length parameter. *)
		arcVelocity : LREAL;
		(* Acceleration of the arc length parameter. *)
		arcAcceleration : LREAL;
	END_VAR
	VAR_IN_OUT
		(* The position at the specified arc parameter. *)
 {attribute 'GUID' := '54EDED35-5A53-0913-4680-EA5D332AAA4F'}
				position : PositionXYC;
		(* The velocity at the specified dynamic state. *)
 {attribute 'GUID' := 'E037A91B-C1D8-04E4-4DB7-2726DA6E0D41'}
				velocity : TangentXYC;
		(* The acceleration at the specified dynamic state. *)
 {attribute 'GUID' := 'E037A91B-C1D8-04E4-4DB7-2726DA6E0D41'}
				acceleration : TangentXYC;
	END_VAR
END_METHOD

END_FUNCTION_BLOCK

// POUs/Shapes/Geometry3D/Container3D

	{attribute 'c++_compatible'}
	{attribute 'external_name' := 'Container3D_GUID_D77467A5_A491_0C26_7B32_760CC7E0EB33'}
	{attribute 'TcIecLibraryType'}
	{attribute 'no_explicit_call' :='do not call this POU directly'}
	{attribute 'no_assign'}
	FUNCTION_BLOCK Container3D EXTENDS Geometry3D


	(* Internal method *)
	METHOD FB_init : BOOL
	VAR_INPUT
		(*  if TRUE, the retain variables are initialized (warm start / cold start) *)
		bInitRetains : BOOL;
		(*  if TRUE, the instance afterwards gets moved into the copy code (online change) *)
		bInCopyCode : BOOL;
	END_VAR
END_METHOD


	(* Internal method *)
	{attribute 'hide'}
	METHOD FB_exit : BOOL
	VAR_INPUT
		(*  if TRUE, the exit method is called for exiting an instance that is copied afterwards (online change). *)
		bInCopyCode : BOOL;
	END_VAR
END_METHOD


	(* Add a geometry to the container. *)
	METHOD AddElement : UDINT
	VAR_IN_OUT
		(* The geometry to add. *)
 {attribute 'GUID' := '56994EB0-AB4F-0BCB-4E0E-A36B53A3D853'}
				geometry : Geometry3D;
	END_VAR
END_METHOD


	(* Remove a specified geometry from the container. *)
	METHOD RemoveElement
	VAR_INPUT
		(* Identifier of the geometry to remove. *)
		id : UDINT;
	END_VAR
END_METHOD


	(* Remove all geometries from container. *)
	METHOD Clear
END_METHOD


	(* Get the number of geometry elements in container. *)
	METHOD GetCount : UDINT
END_METHOD

END_FUNCTION_BLOCK

// POUs/Shapes/Geometry3D/Extrude3D

	{attribute 'c++_compatible'}
	{attribute 'external_name' := 'Extrude3D_GUID_9D8CA6AA_6457_0F6A_7F64_4FCB66BC69A8'}
	{attribute 'TcIecLibraryType'}
	{attribute 'no_explicit_call' :='do not call this POU directly'}
	{attribute 'no_assign'}
	FUNCTION_BLOCK Extrude3D EXTENDS Geometry3D


	(* Internal method *)
	METHOD FB_init : BOOL
	VAR_INPUT
		(*  if TRUE, the retain variables are initialized (warm start / cold start) *)
		bInitRetains : BOOL;
		(*  if TRUE, the instance afterwards gets moved into the copy code (online change) *)
		bInCopyCode : BOOL;
	END_VAR
END_METHOD


	(* Internal method *)
	{attribute 'hide'}
	METHOD FB_exit : BOOL
	VAR_INPUT
		(*  if TRUE, the exit method is called for exiting an instance that is copied afterwards (online change). *)
		bInCopyCode : BOOL;
	END_VAR
END_METHOD


	(* Define the extrude geometry with a path and a array of xy-points *)
	METHOD DefineByPath : BOOL
	VAR_IN_OUT
		(* Cross section values *)
 {attribute 'GUID' := 'D1D75488-37B1-0155-53AF-A9A9BDBB4FFD'}
				PointerToCrossSection : POINTER TO PositionXY;
	END_VAR
	VAR_INPUT
		(* Number of cross section points *)
		NumberOfCrossSectionPoints : UDINT;
	END_VAR
	VAR_IN_OUT
		(* The path *)
 {attribute 'GUID' := '656641C4-F1C9-0188-7114-C4D7E12391DF'}
				Path : PathXYZ;
	END_VAR
	VAR_INPUT
		(* Number of path points *)
		NumberOfPathPoints : UDINT;
	END_VAR
END_METHOD

END_FUNCTION_BLOCK

// POUs/Paths/Components/PathXYZ

	{attribute 'c++_compatible'}
	{attribute 'external_name' := 'PathXYZ_GUID_656641C4_F1C9_0188_7114_C4D7E12391DF'}
	{attribute 'TcIecLibraryType'}
	{attribute 'no_explicit_call' :='do not call this POU directly'}
	{attribute 'no_assign'}
	(* A path in the xy-plane with an additional orientation at every path position. *)
	FUNCTION_BLOCK PathXYZ EXTENDS IPlcPath3D


	(* Internal method *)
	{attribute 'hide'}
	METHOD FB_init : BOOL
	VAR_INPUT
		(*  if TRUE, the retain variables are initialized (warm start / cold start) *)
		bInitRetains : BOOL;
		(*  if TRUE, the instance afterwards gets moved into the copy code (online change) *)
		bInCopyCode : BOOL;
	END_VAR
END_METHOD


	(* Internal method *)
	{attribute 'hide'}
	METHOD FB_exit : BOOL
	VAR_INPUT
		(*  if TRUE, the exit method is called for exiting an instance that is copied afterwards (online change). *)
		bInCopyCode : BOOL;
	END_VAR
END_METHOD


	(* Append a smooth transition from the current end of the path
				    to the specified position. *)
	METHOD AppendPosition
	VAR_IN_OUT
		(* The position to append. *)
 {attribute 'GUID' := '6D9DE39A-582F-0FB5-796C-F5BBE97EF7B7'}
				position : Position3D;
	END_VAR
END_METHOD


	(* Append a smooth transition from the current end of the path
				    to the specified position. *)
	METHOD AppendPositionXYZ
	VAR_INPUT
		(* x-component of the position to append. *)
		x : LREAL;
		(* y-component of the position to append. *)
		y : LREAL;
		(* z-component of the position to append. *)
		c : LREAL;
	END_VAR
END_METHOD


	(* Append a line to this path. *)
	METHOD AppendLine
	VAR_IN_OUT
		(* Start position of the line. *)
 {attribute 'GUID' := '6D9DE39A-582F-0FB5-796C-F5BBE97EF7B7'}
				startPos : Position3D;
		(* End position of the line. *)
 {attribute 'GUID' := '6D9DE39A-582F-0FB5-796C-F5BBE97EF7B7'}
				endPos : Position3D;
	END_VAR
END_METHOD


	(* Append a smooth transition from the current end of the path
				    to the specified position. *)
	METHOD AppendLineXYZ
	VAR_INPUT
		(* x-component of the start position. *)
		x0 : LREAL;
		(* y-component of the start position. *)
		y0 : LREAL;
		(* z-component of the start position. *)
		z0 : LREAL;
		(* x-component of the end position. *)
		x1 : LREAL;
		(* y-component of the end position. *)
		y1 : LREAL;
		(* z-component of the end position. *)
		z1 : LREAL;
	END_VAR
END_METHOD


	(* Append a circle to this path. *)
	METHOD AppendCircle
	VAR_IN_OUT
		(* Start position of the circle. *)
 {attribute 'GUID' := '6D9DE39A-582F-0FB5-796C-F5BBE97EF7B7'}
				startPos : Position3D;
		(* End position of the circle. *)
 {attribute 'GUID' := '6D9DE39A-582F-0FB5-796C-F5BBE97EF7B7'}
				endPos : Position3D;
		(* Center of the circle. *)
 {attribute 'GUID' := 'D1D75488-37B1-0155-53AF-A9A9BDBB4FFD'}
				center : PositionXY;
	END_VAR
	VAR_INPUT
		(* Set whether the circle runs clockwise or counter-clockwise. *)
		clockwise : BOOL;
	END_VAR
END_METHOD


	(* Append a smooth transition from the current end of the path
				    to the specified position with tangent. *)
	METHOD AppendPositionTangent
	VAR_IN_OUT
		(* The position to append. *)
 {attribute 'GUID' := '6D9DE39A-582F-0FB5-796C-F5BBE97EF7B7'}
				position : Position3D;
		(* The tangent to append *)
 {attribute 'GUID' := 'B2E383A0-A70D-05BB-6EF1-4EF1FE579E25'}
				tangent : Tangent3D;
	END_VAR
END_METHOD


	(* Get the start position of the path. *)
	METHOD GetStartPosition
	VAR_IN_OUT
		(* The current start position of the path. *)
 {attribute 'GUID' := '6D9DE39A-582F-0FB5-796C-F5BBE97EF7B7'}
				startPosition : Position3D;
	END_VAR
END_METHOD


	(* Get the end position of the segment. *)
	METHOD GetEndPosition
	VAR_IN_OUT
		(* The current end position of the segment. *)
 {attribute 'GUID' := '6D9DE39A-582F-0FB5-796C-F5BBE97EF7B7'}
				endPosition : Position3D;
	END_VAR
END_METHOD


	(* Get a position on the path at a specific arclength value. *)
	METHOD GetPositionAt
	VAR_INPUT
		(* Arc length value where the position is evaluated. *)
		arcLength : LREAL;
	END_VAR
	VAR_IN_OUT
		(* The position at the specified arc parameter. *)
 {attribute 'GUID' := '6D9DE39A-582F-0FB5-796C-F5BBE97EF7B7'}
				position : Position3D;
	END_VAR
END_METHOD


	(* Get the dynamic information when moving along a path
				    with specific arclength value and dynamic changes. *)
	METHOD GetStateAt
	VAR_INPUT
		(* Arc length value where the position is evaluated. *)
		arcLength : LREAL;
		(* Velocity of the arc length parameter. *)
		arcVelocity : LREAL;
		(* Acceleration of the arc length parameter. *)
		arcAcceleration : LREAL;
	END_VAR
	VAR_IN_OUT
		(* The position at the specified arc parameter. *)
 {attribute 'GUID' := '6D9DE39A-582F-0FB5-796C-F5BBE97EF7B7'}
				position : Position3D;
		(* The velocity at the specified dynamic state. *)
 {attribute 'GUID' := 'B2E383A0-A70D-05BB-6EF1-4EF1FE579E25'}
				velocity : Tangent3D;
		(* The acceleration at the specified dynamic state. *)
 {attribute 'GUID' := 'B2E383A0-A70D-05BB-6EF1-4EF1FE579E25'}
				acceleration : Tangent3D;
	END_VAR
END_METHOD

END_FUNCTION_BLOCK

// POUs/Paths/Components/PathXY

	{attribute 'c++_compatible'}
	{attribute 'external_name' := 'PathXY_GUID_8281DBBF_9A4E_0F66_5E0A_7628DD65B1E6'}
	{attribute 'TcIecLibraryType'}
	{attribute 'no_explicit_call' :='do not call this POU directly'}
	{attribute 'no_assign'}
	(* A path in the xy-plane. *)
	FUNCTION_BLOCK PathXY EXTENDS IPlcPath2D


	(* Internal method *)
	{attribute 'hide'}
	METHOD FB_init : BOOL
	VAR_INPUT
		(*  if TRUE, the retain variables are initialized (warm start / cold start) *)
		bInitRetains : BOOL;
		(*  if TRUE, the instance afterwards gets moved into the copy code (online change) *)
		bInCopyCode : BOOL;
	END_VAR
END_METHOD


	(* Internal method *)
	{attribute 'hide'}
	METHOD FB_exit : BOOL
	VAR_INPUT
		(*  if TRUE, the exit method is called for exiting an instance that is copied afterwards (online change). *)
		bInCopyCode : BOOL;
	END_VAR
END_METHOD


	(* Append a smooth transition from the current end of the path
				    to the specified position. *)
	METHOD AppendPosition
	VAR_IN_OUT
		(* The position to append. *)
 {attribute 'GUID' := 'D1D75488-37B1-0155-53AF-A9A9BDBB4FFD'}
				position : PositionXY;
	END_VAR
END_METHOD


	(* Append a smooth transition from the current end of the path
				    to the specified position. *)
	METHOD AppendPositionXY
	VAR_INPUT
		(* x-component of the position to append. *)
		x : LREAL;
		(* y-component of the position to append. *)
		y : LREAL;
	END_VAR
END_METHOD


	(* Append a line to this path. *)
	METHOD AppendLine
	VAR_IN_OUT
		(* Start position of the line. *)
 {attribute 'GUID' := 'D1D75488-37B1-0155-53AF-A9A9BDBB4FFD'}
				startPos : PositionXY;
		(* End position of the line. *)
 {attribute 'GUID' := 'D1D75488-37B1-0155-53AF-A9A9BDBB4FFD'}
				endPos : PositionXY;
	END_VAR
END_METHOD


	(* Append a circle to this path. *)
	METHOD AppendCircle
	VAR_IN_OUT
		(* Start position of the circle. *)
 {attribute 'GUID' := 'D1D75488-37B1-0155-53AF-A9A9BDBB4FFD'}
				startPos : PositionXY;
		(* End position of the circle. *)
 {attribute 'GUID' := 'D1D75488-37B1-0155-53AF-A9A9BDBB4FFD'}
				endPos : PositionXY;
		(* Center of the circle. *)
 {attribute 'GUID' := 'D1D75488-37B1-0155-53AF-A9A9BDBB4FFD'}
				center : PositionXY;
	END_VAR
	VAR_INPUT
		(* Set whether the circle runs clockwise or counter-clockwise. *)
		clockwise : BOOL;
	END_VAR
END_METHOD


	(* Get the start position of the path. *)
	METHOD GetStartPosition
	VAR_IN_OUT
		(* The current start position of the path. *)
 {attribute 'GUID' := 'D1D75488-37B1-0155-53AF-A9A9BDBB4FFD'}
				startPosition : PositionXY;
	END_VAR
END_METHOD


	(* Get the end position of the segment. *)
	METHOD GetEndPosition
	VAR_IN_OUT
		(* The current end position of the segment. *)
 {attribute 'GUID' := 'D1D75488-37B1-0155-53AF-A9A9BDBB4FFD'}
				endPosition : PositionXY;
	END_VAR
END_METHOD


	(* Get a position on the path at a specific arclength value. *)
	METHOD GetPositionAt
	VAR_INPUT
		(* Arc length value where the position is evaluated. *)
		arcLength : LREAL;
	END_VAR
	VAR_IN_OUT
		(* The position at the specified arc parameter. *)
 {attribute 'GUID' := 'D1D75488-37B1-0155-53AF-A9A9BDBB4FFD'}
				position : PositionXY;
	END_VAR
END_METHOD


	(* Get the dynamic information when moving along a path
				    with specific arclength value and dynamic changes. *)
	METHOD GetStateAt
	VAR_INPUT
		(* Arc length value where the position is evaluated. *)
		arcLength : LREAL;
		(* Velocity of the arc length parameter. *)
		arcVelocity : LREAL;
		(* Acceleration of the arc length parameter. *)
		arcAcceleration : LREAL;
	END_VAR
	VAR_IN_OUT
		(* The position at the specified arc parameter. *)
 {attribute 'GUID' := 'D1D75488-37B1-0155-53AF-A9A9BDBB4FFD'}
				position : PositionXY;
		(* The velocity at the specified dynamic state. *)
 {attribute 'GUID' := '619D5D7D-53EC-0B73-54D5-FB9C43AFDE82'}
				velocity : TangentXY;
		(* The acceleration at the specified dynamic state. *)
 {attribute 'GUID' := '619D5D7D-53EC-0B73-54D5-FB9C43AFDE82'}
				acceleration : TangentXY;
	END_VAR
END_METHOD

END_FUNCTION_BLOCK

// POUs/Shapes/Geometry2D/1D/Line2D

	{attribute 'c++_compatible'}
	{attribute 'external_name' := 'Line2D_GUID_9608B9AC_4BC5_07DF_520D_07E1D5EFD5C4'}
	{attribute 'TcIecLibraryType'}
	{attribute 'no_explicit_call' :='do not call this POU directly'}
	{attribute 'no_assign'}
	(* 2D Geometry Line *)
	FUNCTION_BLOCK Line2D EXTENDS Geometry2D


	(* Internal method *)
	METHOD FB_init : BOOL
	VAR_INPUT
		(*  if TRUE, the retain variables are initialized (warm start / cold start) *)
		bInitRetains : BOOL;
		(*  if TRUE, the instance afterwards gets moved into the copy code (online change) *)
		bInCopyCode : BOOL;
	END_VAR
END_METHOD


	(* Internal method *)
	{attribute 'hide'}
	METHOD FB_exit : BOOL
	VAR_INPUT
		(*  if TRUE, the exit method is called for exiting an instance that is copied afterwards (online change). *)
		bInCopyCode : BOOL;
	END_VAR
END_METHOD


	(* Define a line by two positions. *)
	METHOD DefineByPositions
	VAR_IN_OUT
		(* 1st position on the line to define. *)
 {attribute 'GUID' := 'D1D75488-37B1-0155-53AF-A9A9BDBB4FFD'}
				position0 : PositionXY;
		(* 2nd position on the line to define. *)
 {attribute 'GUID' := 'D1D75488-37B1-0155-53AF-A9A9BDBB4FFD'}
				position1 : PositionXY;
	END_VAR
END_METHOD


	(* Define a line by a position on the line and its direction. *)
	METHOD DefineByDirection
	VAR_IN_OUT
		(* Position on the line *)
 {attribute 'GUID' := 'D1D75488-37B1-0155-53AF-A9A9BDBB4FFD'}
				position : PositionXY;
		(* Direction of the line *)
 {attribute 'GUID' := '619D5D7D-53EC-0B73-54D5-FB9C43AFDE82'}
				direction : TangentXY;
	END_VAR
END_METHOD


	(* Set the direction of the line. *)
	METHOD SetDirection
	VAR_IN_OUT
		(* The direction to set. *)
 {attribute 'GUID' := '619D5D7D-53EC-0B73-54D5-FB9C43AFDE82'}
				direction : TangentXY;
	END_VAR
END_METHOD


	(* Get the direction of the line. *)
	METHOD GetDirection
	VAR_IN_OUT
		(* The current direction of the line. *)
 {attribute 'GUID' := '619D5D7D-53EC-0B73-54D5-FB9C43AFDE82'}
				direction : TangentXY;
	END_VAR
END_METHOD


	(* Get a position on the line at a specific arclength value. *)
	METHOD GetPositionAt
	VAR_INPUT
		(* Arc length value where the position is evaluated. *)
		arcLength : LREAL;
	END_VAR
	VAR_IN_OUT
		(* The position at the specified arc parameter. *)
 {attribute 'GUID' := '54EDED35-5A53-0913-4680-EA5D332AAA4F'}
				position : PositionXYC;
	END_VAR
END_METHOD

END_FUNCTION_BLOCK

// POUs/Shapes/Geometry2D/1D/Segment2D

	{attribute 'c++_compatible'}
	{attribute 'external_name' := 'Segment2D_GUID_F7F959A9_4A43_0FC1_515B_72317DA3461E'}
	{attribute 'TcIecLibraryType'}
	{attribute 'no_explicit_call' :='do not call this POU directly'}
	{attribute 'no_assign'}
	FUNCTION_BLOCK Segment2D EXTENDS Geometry2D


	(* Internal method *)
	METHOD FB_init : BOOL
	VAR_INPUT
		(*  if TRUE, the retain variables are initialized (warm start / cold start) *)
		bInitRetains : BOOL;
		(*  if TRUE, the instance afterwards gets moved into the copy code (online change) *)
		bInCopyCode : BOOL;
	END_VAR
END_METHOD


	(* Internal method *)
	{attribute 'hide'}
	METHOD FB_exit : BOOL
	VAR_INPUT
		(*  if TRUE, the exit method is called for exiting an instance that is copied afterwards (online change). *)
		bInCopyCode : BOOL;
	END_VAR
END_METHOD


	(* Set the start position of the segment. *)
	METHOD SetStartPosition
	VAR_IN_OUT
		(* Start position of the segment to set. *)
 {attribute 'GUID' := 'D1D75488-37B1-0155-53AF-A9A9BDBB4FFD'}
				startPos : PositionXY;
	END_VAR
END_METHOD


	(* Set the start position of the segment. *)
	METHOD SetStartPositionXY
	VAR_INPUT
		(* x-component of the start position. *)
		x : LREAL;
		(* y-component of the start position. *)
		y : LREAL;
	END_VAR
END_METHOD


	(* Set the end position of the segment. *)
	METHOD SetEndPosition
	VAR_IN_OUT
		(* End position of the segment to set. *)
 {attribute 'GUID' := 'D1D75488-37B1-0155-53AF-A9A9BDBB4FFD'}
				endPos : PositionXY;
	END_VAR
END_METHOD


	(* Set the end position of the segment. *)
	METHOD SetEndPositionXY
	VAR_INPUT
		(* x-component of the end position. *)
		x : LREAL;
		(* y-component of the end position. *)
		y : LREAL;
	END_VAR
END_METHOD


	(* Get the x-component of the segment length in respect to the root coordinate system. *)
	METHOD Get_dX : LREAL
END_METHOD


	(* Get the y-component of the segment length in respect to the root coordinate system. *)
	METHOD Get_dY : LREAL
END_METHOD


	(* Get the length of the segment. *)
	METHOD GetLength : LREAL
END_METHOD


	(* Get the start position of the segment. *)
	METHOD GetStartPosition
	VAR_IN_OUT
		(* The current start position of the segment. *)
 {attribute 'GUID' := 'D1D75488-37B1-0155-53AF-A9A9BDBB4FFD'}
				startPosition : PositionXY;
	END_VAR
END_METHOD


	(* Get the end position of the segment. *)
	METHOD GetEndPosition
	VAR_IN_OUT
		(* The current end position of the segment. *)
 {attribute 'GUID' := 'D1D75488-37B1-0155-53AF-A9A9BDBB4FFD'}
				endPosition : PositionXY;
	END_VAR
END_METHOD


	(* Get the direction of the segment. *)
	METHOD GetDirection
	VAR_IN_OUT
		(* The current direction of the segment. *)
 {attribute 'GUID' := '619D5D7D-53EC-0B73-54D5-FB9C43AFDE82'}
				direction : TangentXY;
	END_VAR
END_METHOD


	(* Get a position on the segment at a specific arclength value. *)
	METHOD GetPositionAt
	VAR_INPUT
		(* Arc length value where the position is evaluated. *)
		arcLength : LREAL;
	END_VAR
	VAR_IN_OUT
		(* The position at the specified arc parameter. *)
 {attribute 'GUID' := '54EDED35-5A53-0913-4680-EA5D332AAA4F'}
				position : PositionXYC;
	END_VAR
END_METHOD

END_FUNCTION_BLOCK

// POUs/Shapes/Geometry2D/1D/Circle2D

	{attribute 'c++_compatible'}
	{attribute 'external_name' := 'Circle2D_GUID_A0BE8ADA_46DF_0C08_6381_50015B0A03BF'}
	{attribute 'TcIecLibraryType'}
	{attribute 'no_explicit_call' :='do not call this POU directly'}
	{attribute 'no_assign'}
	FUNCTION_BLOCK Circle2D EXTENDS Geometry2D


	(* Internal method *)
	METHOD FB_init : BOOL
	VAR_INPUT
		(*  if TRUE, the retain variables are initialized (warm start / cold start) *)
		bInitRetains : BOOL;
		(*  if TRUE, the instance afterwards gets moved into the copy code (online change) *)
		bInCopyCode : BOOL;
	END_VAR
END_METHOD


	(* Internal method *)
	{attribute 'hide'}
	METHOD FB_exit : BOOL
	VAR_INPUT
		(*  if TRUE, the exit method is called for exiting an instance that is copied afterwards (online change). *)
		bInCopyCode : BOOL;
	END_VAR
END_METHOD


	(* Get the length of the circle. *)
	METHOD GetLength : LREAL
END_METHOD


	(* Get a position on the circle at a specific arclength value. *)
	METHOD GetPositionAt
	VAR_INPUT
		(* Arc length value where the position is evaluated. *)
		arcLength : LREAL;
	END_VAR
	VAR_IN_OUT
		(* The position at the specified arc parameter. *)
 {attribute 'GUID' := '54EDED35-5A53-0913-4680-EA5D332AAA4F'}
				position : PositionXYC;
	END_VAR
END_METHOD


	PROPERTY radius : LREAL
GET
END_GET
SET
END_SET
END_PROPERTY

END_FUNCTION_BLOCK

// POUs/Shapes/Geometry2D/2D/Disc2D

	{attribute 'c++_compatible'}
	{attribute 'external_name' := 'Disc2D_GUID_5D49F634_D804_05FE_7BC3_DB605F1B0693'}
	{attribute 'TcIecLibraryType'}
	{attribute 'no_explicit_call' :='do not call this POU directly'}
	{attribute 'no_assign'}
	FUNCTION_BLOCK Disc2D EXTENDS Geometry2D


	(* Internal method *)
	METHOD FB_init : BOOL
	VAR_INPUT
		(*  if TRUE, the retain variables are initialized (warm start / cold start) *)
		bInitRetains : BOOL;
		(*  if TRUE, the instance afterwards gets moved into the copy code (online change) *)
		bInCopyCode : BOOL;
	END_VAR
END_METHOD


	(* Internal method *)
	{attribute 'hide'}
	METHOD FB_exit : BOOL
	VAR_INPUT
		(*  if TRUE, the exit method is called for exiting an instance that is copied afterwards (online change). *)
		bInCopyCode : BOOL;
	END_VAR
END_METHOD


	(* Get the area of the disc. *)
	METHOD GetArea : LREAL
END_METHOD


	PROPERTY radius : LREAL
GET
END_GET
SET
END_SET
END_PROPERTY

END_FUNCTION_BLOCK

// POUs/Shapes/Geometry2D/2D/Rectangle2D

	{attribute 'c++_compatible'}
	{attribute 'external_name' := 'Rectangle2D_GUID_736BC5A9_5C61_09B6_601B_606942FC2981'}
	{attribute 'TcIecLibraryType'}
	{attribute 'no_explicit_call' :='do not call this POU directly'}
	{attribute 'no_assign'}
	FUNCTION_BLOCK Rectangle2D EXTENDS Geometry2D


	(* Internal method *)
	METHOD FB_init : BOOL
	VAR_INPUT
		(*  if TRUE, the retain variables are initialized (warm start / cold start) *)
		bInitRetains : BOOL;
		(*  if TRUE, the instance afterwards gets moved into the copy code (online change) *)
		bInCopyCode : BOOL;
	END_VAR
END_METHOD


	(* Internal method *)
	{attribute 'hide'}
	METHOD FB_exit : BOOL
	VAR_INPUT
		(*  if TRUE, the exit method is called for exiting an instance that is copied afterwards (online change). *)
		bInCopyCode : BOOL;
	END_VAR
END_METHOD


	(* Set the dimensions of the rectangle. *)
	METHOD SetDimensions
	VAR_INPUT
		(* The width of the rectangle to set. *)
		width : LREAL;
		(* The height of the rectangle to set. *)
		height : LREAL;
	END_VAR
END_METHOD


	(* Get the area of the rectangle. *)
	METHOD GetArea : LREAL
END_METHOD


	PROPERTY width : LREAL
GET
END_GET
SET
END_SET
END_PROPERTY


	PROPERTY height : LREAL
GET
END_GET
SET
END_SET
END_PROPERTY

END_FUNCTION_BLOCK

// POUs/Shapes/Geometry2D/Functions/CheckCollision2D

	{attribute 'TcIecLibraryType'}
	{attribute 'external_name' := 'CheckCollision2D_GUID_CDD85A2E_C698_0248_6D59_F851C6A31905'}
	(* Check if two geometries are currently colliding. *)
	FUNCTION CheckCollision2D : BOOL
	VAR_IN_OUT
		geometry0	:	IPlcGeometry2D;	(* 1st input geometry to check for collision. *)
		geometry1	:	IPlcGeometry2D;	(* 2nd input geometry to check of collision. *)
	END_VAR

END_FUNCTION

// POUs/Shapes/Geometry2D/Functions/GetDistance2D

	{attribute 'TcIecLibraryType'}
	{attribute 'external_name' := 'GetDistance2D_GUID_F21721D6_07E3_08DD_5915_F6707318C499'}
	(* Get the distance between two geometries. *)
	FUNCTION GetDistance2D : LREAL
	VAR_IN_OUT
		geometry0	:	IPlcGeometry2D;	(* 1st input geometry to calculate the distance of. *)
		geometry1	:	IPlcGeometry2D;	(* 2nd input geometry to calculate the distance of. *)
	END_VAR

END_FUNCTION

// POUs/Shapes/Geometry2D/Functions/GetLinkingLine2D

	{attribute 'TcIecLibraryType'}
	{attribute 'external_name' := 'GetLinkingLine2D_GUID_B4FC21E9_7515_06B0_7D6B_99EB3A346BCF'}
	(* Get the shortest path between two geometries. *)
	FUNCTION GetLinkingLine2D : BOOL
	VAR_IN_OUT
		geometry0	:	IPlcGeometry2D;	(* 1st input geometry to calculate the linking line for. *)
		geometry1	:	IPlcGeometry2D;	(* 2nd input geometry to calculate the linking line for. *)
		linkingLine	:	Segment2D;	(* Return the resulting linking line. *)
	END_VAR

END_FUNCTION

// POUs/Shapes/Geometry3D/1D/Line3D

	{attribute 'c++_compatible'}
	{attribute 'external_name' := 'Line3D_GUID_9BB6C223_1930_0F23_7B94_62618179CDDF'}
	{attribute 'TcIecLibraryType'}
	{attribute 'no_explicit_call' :='do not call this POU directly'}
	{attribute 'no_assign'}
	(* 3D Geometry Line *)
	FUNCTION_BLOCK Line3D EXTENDS Geometry3D


	(* Internal method *)
	METHOD FB_init : BOOL
	VAR_INPUT
		(*  if TRUE, the retain variables are initialized (warm start / cold start) *)
		bInitRetains : BOOL;
		(*  if TRUE, the instance afterwards gets moved into the copy code (online change) *)
		bInCopyCode : BOOL;
	END_VAR
END_METHOD


	(* Internal method *)
	{attribute 'hide'}
	METHOD FB_exit : BOOL
	VAR_INPUT
		(*  if TRUE, the exit method is called for exiting an instance that is copied afterwards (online change). *)
		bInCopyCode : BOOL;
	END_VAR
END_METHOD


	(* Define a line by two positions. *)
	METHOD DefineByPositions
	VAR_IN_OUT
		(* 1st position on the line to define. *)
 {attribute 'GUID' := '6D9DE39A-582F-0FB5-796C-F5BBE97EF7B7'}
				position0 : Position3D;
		(* 2nd position on the line to define. *)
 {attribute 'GUID' := '6D9DE39A-582F-0FB5-796C-F5BBE97EF7B7'}
				position1 : Position3D;
	END_VAR
END_METHOD


	(* Define a line by a position on the line and its direction. *)
	METHOD DefineByDirection
	VAR_IN_OUT
		(* Position on the line. *)
 {attribute 'GUID' := '6D9DE39A-582F-0FB5-796C-F5BBE97EF7B7'}
				position : Position3D;
		(* Direction of the line. *)
 {attribute 'GUID' := 'B2E383A0-A70D-05BB-6EF1-4EF1FE579E25'}
				direction : Tangent3D;
	END_VAR
END_METHOD


	(* Set the direction of the line. *)
	METHOD SetDirection
	VAR_IN_OUT
		(* The direction to set. *)
 {attribute 'GUID' := 'B2E383A0-A70D-05BB-6EF1-4EF1FE579E25'}
				direction : Tangent3D;
	END_VAR
END_METHOD


	(* Get the direction of the line. *)
	METHOD GetDirection
	VAR_IN_OUT
		(* The current direction of the line. *)
 {attribute 'GUID' := 'B2E383A0-A70D-05BB-6EF1-4EF1FE579E25'}
				direction : Tangent3D;
	END_VAR
END_METHOD


	(* Get a position on the line at a specific arclength value. *)
	METHOD GetPositionAt
	VAR_INPUT
		(* Arc length value where the position is evaluated. *)
		arcLength : LREAL;
	END_VAR
	VAR_IN_OUT
		(* The position at the specified arc parameter. *)
 {attribute 'GUID' := '4DF191CB-C971-05F9-659B-EBBADE382F22'}
				position : PositionSE3;
	END_VAR
END_METHOD

END_FUNCTION_BLOCK

// POUs/Shapes/Geometry3D/1D/Segment3D

	{attribute 'c++_compatible'}
	{attribute 'external_name' := 'Segment3D_GUID_A667D0B1_A6CC_0807_63BD_1DD566E90D8F'}
	{attribute 'TcIecLibraryType'}
	{attribute 'no_explicit_call' :='do not call this POU directly'}
	{attribute 'no_assign'}
	FUNCTION_BLOCK Segment3D EXTENDS Geometry3D


	(* Internal method *)
	METHOD FB_init : BOOL
	VAR_INPUT
		(*  if TRUE, the retain variables are initialized (warm start / cold start) *)
		bInitRetains : BOOL;
		(*  if TRUE, the instance afterwards gets moved into the copy code (online change) *)
		bInCopyCode : BOOL;
	END_VAR
END_METHOD


	(* Internal method *)
	{attribute 'hide'}
	METHOD FB_exit : BOOL
	VAR_INPUT
		(*  if TRUE, the exit method is called for exiting an instance that is copied afterwards (online change). *)
		bInCopyCode : BOOL;
	END_VAR
END_METHOD


	(* Set the start position of the segment. *)
	METHOD SetStartPosition
	VAR_IN_OUT
		(* Start position of the segment to set. *)
 {attribute 'GUID' := '6D9DE39A-582F-0FB5-796C-F5BBE97EF7B7'}
				startPos : Position3D;
	END_VAR
END_METHOD


	(* Set the start position of the segment. *)
	METHOD SetStartPositionXYZ
	VAR_INPUT
		(* x-component of the start position. *)
		x : LREAL;
		(* y-component of the start position. *)
		y : LREAL;
		(* z-component of the start position. *)
		z : LREAL;
	END_VAR
END_METHOD


	(* Set the end position of the segment. *)
	METHOD SetEndPosition
	VAR_IN_OUT
		(* End position of the segment to set. *)
 {attribute 'GUID' := '6D9DE39A-582F-0FB5-796C-F5BBE97EF7B7'}
				endPos : Position3D;
	END_VAR
END_METHOD


	(* Set the end position of the segment. *)
	METHOD SetEndPositionXYZ
	VAR_INPUT
		(* x-component of the end position. *)
		x : LREAL;
		(* y-component of the end position. *)
		y : LREAL;
		(* z-component of the end position. *)
		z : LREAL;
	END_VAR
END_METHOD


	(* Get the x-component of the segment length in respect to the root coordinate system. *)
	METHOD Get_dX : LREAL
END_METHOD


	(* Get the y-component of the segment length in respect to the root coordinate system. *)
	METHOD Get_dY : LREAL
END_METHOD


	(* Get the z-component of the segment length in respect to the root coordinate system. *)
	METHOD Get_dZ : LREAL
END_METHOD


	(* Get the length of the segment. *)
	METHOD GetLength : LREAL
END_METHOD


	(* Get the start position of the segment. *)
	METHOD GetStartPosition
	VAR_IN_OUT
		(* The current start position of the segment. *)
 {attribute 'GUID' := '6D9DE39A-582F-0FB5-796C-F5BBE97EF7B7'}
				startPosition : Position3D;
	END_VAR
END_METHOD


	(* Get the end position of the segment. *)
	METHOD GetEndPosition
	VAR_IN_OUT
		(* The current end position of the segment. *)
 {attribute 'GUID' := '6D9DE39A-582F-0FB5-796C-F5BBE97EF7B7'}
				endPosition : Position3D;
	END_VAR
END_METHOD


	(* Get the direction of the segment. *)
	METHOD GetDirection
	VAR_IN_OUT
		(* The current direction of the segment. *)
 {attribute 'GUID' := 'B2E383A0-A70D-05BB-6EF1-4EF1FE579E25'}
				direction : Tangent3D;
	END_VAR
END_METHOD


	(* Get a position on the segment at a specific arclength value. *)
	METHOD GetPositionAt
	VAR_INPUT
		(* Arc length value where the position is evaluated. *)
		arcLength : LREAL;
	END_VAR
	VAR_IN_OUT
		(* The position at the specified arc parameter. *)
 {attribute 'GUID' := '4DF191CB-C971-05F9-659B-EBBADE382F22'}
				position : PositionSE3;
	END_VAR
END_METHOD

END_FUNCTION_BLOCK

// POUs/Shapes/Geometry3D/1D/Circle3D

	{attribute 'c++_compatible'}
	{attribute 'external_name' := 'Circle3D_GUID_6ED10856_9A22_08B9_7704_8FEF53E0B9E2'}
	{attribute 'TcIecLibraryType'}
	{attribute 'no_explicit_call' :='do not call this POU directly'}
	{attribute 'no_assign'}
	FUNCTION_BLOCK Circle3D EXTENDS Geometry3D


	(* Internal method *)
	METHOD FB_init : BOOL
	VAR_INPUT
		(*  if TRUE, the retain variables are initialized (warm start / cold start) *)
		bInitRetains : BOOL;
		(*  if TRUE, the instance afterwards gets moved into the copy code (online change) *)
		bInCopyCode : BOOL;
	END_VAR
END_METHOD


	(* Internal method *)
	{attribute 'hide'}
	METHOD FB_exit : BOOL
	VAR_INPUT
		(*  if TRUE, the exit method is called for exiting an instance that is copied afterwards (online change). *)
		bInCopyCode : BOOL;
	END_VAR
END_METHOD


	(* Set the normal vector of the circle. *)
	METHOD SetNormal
	VAR_IN_OUT
		(* Normal vector to set. *)
 {attribute 'GUID' := 'B2E383A0-A70D-05BB-6EF1-4EF1FE579E25'}
				normal : Tangent3D;
	END_VAR
END_METHOD


	(* Get the length of the circle. *)
	METHOD GetLength : LREAL
END_METHOD


	(* Get the normal vector of the circle. *)
	METHOD GetNormal
	VAR
		(* The current normal vector of the circle. *)
 {attribute 'GUID' := 'B2E383A0-A70D-05BB-6EF1-4EF1FE579E25'}
				normal : Tangent3D;
	END_VAR
END_METHOD


	(* Get a position on the circle at a specific arclength value. *)
	METHOD GetPositionAt
	VAR_INPUT
		(* Arc length value where the position is evaluated. *)
		arcLength : LREAL;
	END_VAR
	VAR_IN_OUT
		(* The position at the specified arc parameter. *)
 {attribute 'GUID' := '4DF191CB-C971-05F9-659B-EBBADE382F22'}
				position : PositionSE3;
	END_VAR
END_METHOD


	PROPERTY radius : LREAL
GET
END_GET
SET
END_SET
END_PROPERTY

END_FUNCTION_BLOCK

// POUs/Shapes/Geometry3D/2D/Plane3D

	{attribute 'c++_compatible'}
	{attribute 'external_name' := 'Plane3D_GUID_9FE1EA27_93AF_0368_5C1A_D79F7E5FECF7'}
	{attribute 'TcIecLibraryType'}
	{attribute 'no_explicit_call' :='do not call this POU directly'}
	{attribute 'no_assign'}
	FUNCTION_BLOCK Plane3D EXTENDS Geometry3D


	(* Internal method *)
	METHOD FB_init : BOOL
	VAR_INPUT
		(*  if TRUE, the retain variables are initialized (warm start / cold start) *)
		bInitRetains : BOOL;
		(*  if TRUE, the instance afterwards gets moved into the copy code (online change) *)
		bInCopyCode : BOOL;
	END_VAR
END_METHOD


	(* Internal method *)
	{attribute 'hide'}
	METHOD FB_exit : BOOL
	VAR_INPUT
		(*  if TRUE, the exit method is called for exiting an instance that is copied afterwards (online change). *)
		bInCopyCode : BOOL;
	END_VAR
END_METHOD


	(* Set the normal of the plane. *)
	METHOD SetNormal
	VAR_IN_OUT
		(* The normal vector to set. *)
 {attribute 'GUID' := 'B2E383A0-A70D-05BB-6EF1-4EF1FE579E25'}
				normal : Tangent3D;
	END_VAR
END_METHOD


	(* Get the normal vector of the plane. *)
	METHOD GetNormal
	VAR
		(* The current normal vector of the plane. *)
 {attribute 'GUID' := 'B2E383A0-A70D-05BB-6EF1-4EF1FE579E25'}
				normal : Tangent3D;
	END_VAR
END_METHOD

END_FUNCTION_BLOCK

// POUs/Shapes/Geometry3D/2D/Disc3D

	{attribute 'c++_compatible'}
	{attribute 'external_name' := 'Disc3D_GUID_055F04F8_014C_0F7C_56B4_802D1F5982B5'}
	{attribute 'TcIecLibraryType'}
	{attribute 'no_explicit_call' :='do not call this POU directly'}
	{attribute 'no_assign'}
	FUNCTION_BLOCK Disc3D EXTENDS Geometry3D


	(* Internal method *)
	METHOD FB_init : BOOL
	VAR_INPUT
		(*  if TRUE, the retain variables are initialized (warm start / cold start) *)
		bInitRetains : BOOL;
		(*  if TRUE, the instance afterwards gets moved into the copy code (online change) *)
		bInCopyCode : BOOL;
	END_VAR
END_METHOD


	(* Internal method *)
	{attribute 'hide'}
	METHOD FB_exit : BOOL
	VAR_INPUT
		(*  if TRUE, the exit method is called for exiting an instance that is copied afterwards (online change). *)
		bInCopyCode : BOOL;
	END_VAR
END_METHOD


	(* Set the normal vector of the disc. *)
	METHOD SetNormal
	VAR_IN_OUT
		(* The normal to set. *)
 {attribute 'GUID' := 'B2E383A0-A70D-05BB-6EF1-4EF1FE579E25'}
				normal : Tangent3D;
	END_VAR
END_METHOD


	(* Get the normal vector of the disc. *)
	METHOD GetNormal
	VAR
		(* The current normal vector of the disc. *)
 {attribute 'GUID' := 'B2E383A0-A70D-05BB-6EF1-4EF1FE579E25'}
				normal : Tangent3D;
	END_VAR
END_METHOD


	(* Get the area of the disc. *)
	METHOD GetArea : LREAL
END_METHOD


	PROPERTY radius : LREAL
GET
END_GET
SET
END_SET
END_PROPERTY

END_FUNCTION_BLOCK

// POUs/Shapes/Geometry3D/2D/Rectangle3D

	{attribute 'c++_compatible'}
	{attribute 'external_name' := 'Rectangle3D_GUID_57D197B5_D3CA_07EB_74B2_2F99D5DE228B'}
	{attribute 'TcIecLibraryType'}
	{attribute 'no_explicit_call' :='do not call this POU directly'}
	{attribute 'no_assign'}
	FUNCTION_BLOCK Rectangle3D EXTENDS Geometry3D


	(* Internal method *)
	METHOD FB_init : BOOL
	VAR_INPUT
		(*  if TRUE, the retain variables are initialized (warm start / cold start) *)
		bInitRetains : BOOL;
		(*  if TRUE, the instance afterwards gets moved into the copy code (online change) *)
		bInCopyCode : BOOL;
	END_VAR
END_METHOD


	(* Internal method *)
	{attribute 'hide'}
	METHOD FB_exit : BOOL
	VAR_INPUT
		(*  if TRUE, the exit method is called for exiting an instance that is copied afterwards (online change). *)
		bInCopyCode : BOOL;
	END_VAR
END_METHOD


	(* Set the dimensions of the rectangle. *)
	METHOD SetDimensions
	VAR_INPUT
		(* The width of the rectangle to set. *)
		width : LREAL;
		(* The height of the rectangle to set. *)
		height : LREAL;
	END_VAR
END_METHOD


	(* Get the area of the rectangle. *)
	METHOD GetArea : LREAL
END_METHOD


	PROPERTY width : LREAL
GET
END_GET
SET
END_SET
END_PROPERTY


	PROPERTY height : LREAL
GET
END_GET
SET
END_SET
END_PROPERTY

END_FUNCTION_BLOCK

// POUs/Shapes/Geometry3D/3D/Sphere3D

	{attribute 'c++_compatible'}
	{attribute 'external_name' := 'Sphere3D_GUID_AD399A98_8D50_02FA_67D4_5110C1F642E9'}
	{attribute 'TcIecLibraryType'}
	{attribute 'no_explicit_call' :='do not call this POU directly'}
	{attribute 'no_assign'}
	FUNCTION_BLOCK Sphere3D EXTENDS Geometry3D


	(* Internal method *)
	METHOD FB_init : BOOL
	VAR_INPUT
		(*  if TRUE, the retain variables are initialized (warm start / cold start) *)
		bInitRetains : BOOL;
		(*  if TRUE, the instance afterwards gets moved into the copy code (online change) *)
		bInCopyCode : BOOL;
	END_VAR
END_METHOD


	(* Internal method *)
	{attribute 'hide'}
	METHOD FB_exit : BOOL
	VAR_INPUT
		(*  if TRUE, the exit method is called for exiting an instance that is copied afterwards (online change). *)
		bInCopyCode : BOOL;
	END_VAR
END_METHOD


	(* Get the volume of the sphere. *)
	METHOD GetVolume : LREAL
END_METHOD


	PROPERTY radius : LREAL
GET
END_GET
SET
END_SET
END_PROPERTY

END_FUNCTION_BLOCK

// POUs/Shapes/Geometry3D/3D/Cuboid3D

	{attribute 'c++_compatible'}
	{attribute 'external_name' := 'Cuboid3D_GUID_5F230E1B_F8BF_04CD_5DF3_8FCBF02AC641'}
	{attribute 'TcIecLibraryType'}
	{attribute 'no_explicit_call' :='do not call this POU directly'}
	{attribute 'no_assign'}
	FUNCTION_BLOCK Cuboid3D EXTENDS Geometry3D


	(* Internal method *)
	METHOD FB_init : BOOL
	VAR_INPUT
		(* if TRUE, the retain variables are initialized (warm start / cold start) *)
		bInitRetains : BOOL;
		(* if TRUE, the instance afterwards gets moved into the copy code (online change) *)
		bInCopyCode : BOOL;
	END_VAR
END_METHOD


	(* Internal method *)
	{attribute 'hide'}
	METHOD FB_exit : BOOL
	VAR_INPUT
		(* if TRUE, the exit method is called for exiting an instance that is copied afterwards (online change). *)
		bInCopyCode : BOOL;
	END_VAR
END_METHOD


	(* Set the dimensions of the cuboid. *)
	METHOD SetDimensions
	VAR_INPUT
		(* local x-component *)
		length : LREAL;
		(* local y-component *)
		width : LREAL;
		(* local z-component *)
		height : LREAL;
	END_VAR
END_METHOD


	(* Get the volume of the cuboid. *)
	METHOD GetVolume : LREAL
END_METHOD


	PROPERTY length : LREAL
GET
END_GET
SET
END_SET
END_PROPERTY


	PROPERTY width : LREAL
GET
END_GET
SET
END_SET
END_PROPERTY


	PROPERTY height : LREAL
GET
END_GET
SET
END_SET
END_PROPERTY

END_FUNCTION_BLOCK

// POUs/Shapes/Geometry3D/3D/Cylinder3D

	{attribute 'c++_compatible'}
	{attribute 'external_name' := 'Cylinder3D_GUID_3BBD5421_DF97_0C2F_43A0_3100D18296E6'}
	{attribute 'TcIecLibraryType'}
	{attribute 'no_explicit_call' :='do not call this POU directly'}
	{attribute 'no_assign'}
	FUNCTION_BLOCK Cylinder3D EXTENDS Geometry3D


	(* Internal method *)
	METHOD FB_init : BOOL
	VAR_INPUT
		(* if TRUE, the retain variables are initialized (warm start / cold start) *)
		bInitRetains : BOOL;
		(* if TRUE, the instance afterwards gets moved into the copy code (online change) *)
		bInCopyCode : BOOL;
	END_VAR
END_METHOD


	(* Internal method *)
	{attribute 'hide'}
	METHOD FB_exit : BOOL
	VAR_INPUT
		(* if TRUE, the exit method is called for exiting an instance that is copied afterwards (online change). *)
		bInCopyCode : BOOL;
	END_VAR
END_METHOD


	(* Set the dimensions of the cylinder. *)
	METHOD SetDimensions
	VAR_INPUT
		(* The radius to set. *)
		radius : LREAL;
		(* The height to set. *)
		height : LREAL;
	END_VAR
END_METHOD


	(* Get the volume of the cylinder. *)
	METHOD GetVolume : LREAL
END_METHOD


	PROPERTY radius : LREAL
GET
END_GET
SET
END_SET
END_PROPERTY


	PROPERTY height : LREAL
GET
END_GET
SET
END_SET
END_PROPERTY

END_FUNCTION_BLOCK

// POUs/Shapes/Geometry3D/Functions/CheckCollision3D

	{attribute 'TcIecLibraryType'}
	{attribute 'external_name' := 'CheckCollision3D_GUID_585D568A_B3EB_0D10_780F_314A51F9EC73'}
	(* Check if two geometries are currently colliding. *)
	FUNCTION CheckCollision3D : BOOL
	VAR_IN_OUT
		geometry0	:	IPlcGeometry3D;	(* 1st input geometry to check for collision. *)
		geometry1	:	IPlcGeometry3D;	(* 2nd input geometry to check of collision. *)
	END_VAR

END_FUNCTION

// POUs/Shapes/Geometry3D/Functions/GetDistance3D

	{attribute 'TcIecLibraryType'}
	{attribute 'external_name' := 'GetDistance3D_GUID_ABE4689F_2431_0A14_5738_E112ED55B9CB'}
	(* Get the distance between two geometries. *)
	FUNCTION GetDistance3D : LREAL
	VAR_IN_OUT
		geometry0	:	IPlcGeometry3D;	(* 1st input geometry to calculate the distance of. *)
		geometry1	:	IPlcGeometry3D;	(* 2nd input geometry to calculate the distance of. *)
	END_VAR

END_FUNCTION

// POUs/Shapes/Geometry3D/Functions/GetLinkingLine3D

	{attribute 'TcIecLibraryType'}
	{attribute 'external_name' := 'GetLinkingLine3D_GUID_C8D96394_A4FE_05C0_64F5_88840DC99209'}
	(* Get the shortest path between two geometries. *)
	FUNCTION GetLinkingLine3D : BOOL
	VAR_IN_OUT
		geometry0	:	IPlcGeometry3D;	(* 1st input geometry to calculate the linking line for. *)
		geometry1	:	IPlcGeometry3D;	(* 2nd input geometry to calculate the linking line for. *)
		linkingLine	:	Segment3D;	(* Return the resulting linking line. *)
	END_VAR

END_FUNCTION

// POUs/Shapes/Geometry3D/Functions/CreateIntersection2D

	{attribute 'TcIecLibraryType'}
	{attribute 'external_name' := 'CreateIntersection2D_GUID_F404FB79_53C2_0EB8_7BDB_652C1280F58D'}
	(* Create a collection of intersections along a plane definition. *)
	FUNCTION CreateIntersection2D : BOOL
	VAR_IN_OUT
		container3D	:	Container3D;	(* Input container to create the intersections of. *)
		planeFrame	:	PositionSE3;	(* The coordinate frame to indicate the origin of the plane. *)
		container2D	:	Container2D;	(* Return the resulting collection of intersection. *)
	END_VAR

END_FUNCTION
